// TIA Portal project "mixer" (V16)

(* hardware
DEVICE "S7300/ET200M station_1"  S7-300 station
   slot 0: "Rail_0"  Rail  6ES7 390-1***0-0AA0
   slot 2: "PLC_1"  CPU 312  6ES7 312-1AE13-0AB0  V2.6
      slot 0: "MPI interface_1"  X1
*)

// ===== PLC "PLC_1"  CPU 312 =====

VAR_GLOBAL   // PLC tag table "Default tag table"
   "C Start" AT %I0.0 : Bool;
   "C stop" AT %I0.1 : Bool;
   "C ON" AT %M0.0 : Bool;
   "Empty level switch I" AT %I0.4 : Bool;
   "In valve1" AT %Q0.0 : Bool;
   "Lvl of mat A" AT %I0.3 : Bool;
   "In valve2" AT %Q0.1 : Bool;
   "Lvl of mat B" AT %I0.2 : Bool;
   "Agitator-mix- moto" AT %Q0.2 : Bool;
   "Temp Sensor" AT %I0.5 : Bool;
   "Heater" AT %Q0.3 : Bool;
   "out valve" AT %Q0.4 : Bool;
END_VAR

ORGANIZATION_BLOCK "Main"   // OB1, LAD
TITLE = "Main Program Sweep (Cycle)"
{ S7_Optimized_Access := 'FALSE' }
VERSION : 0.1
   VAR_TEMP
      OB1_EV_CLASS : Byte;   // Bits 0-3 = 1 (Coming event), Bits 4-7 = 1 (Event class 1)
      OB1_SCAN_1 : Byte;   // 1 (Cold restart scan 1 of OB 1), 3 (Scan 2-n of OB 1)
      OB1_PRIORITY : Byte;   // Priority of OB Execution
      OB1_OB_NUMBR : Byte;   // 1 (Organization block 1, OB1)
      OB1_RESERVED_1 : Byte;   // Reserved for system
      OB1_RESERVED_2 : Byte;   // Reserved for system
      OB1_PREV_CYCLE : Int;   // Cycle time of previous OB1 scan (milliseconds)
      OB1_MIN_CYCLE : Int;   // Minimum cycle time of OB1 (milliseconds)
      OB1_MAX_CYCLE : Int;   // Maximum cycle time of OB1 (milliseconds)
      OB1_DATE_TIME : Date_And_Time;   // Date and time OB1 started
   END_VAR
BEGIN

REGION Network 1
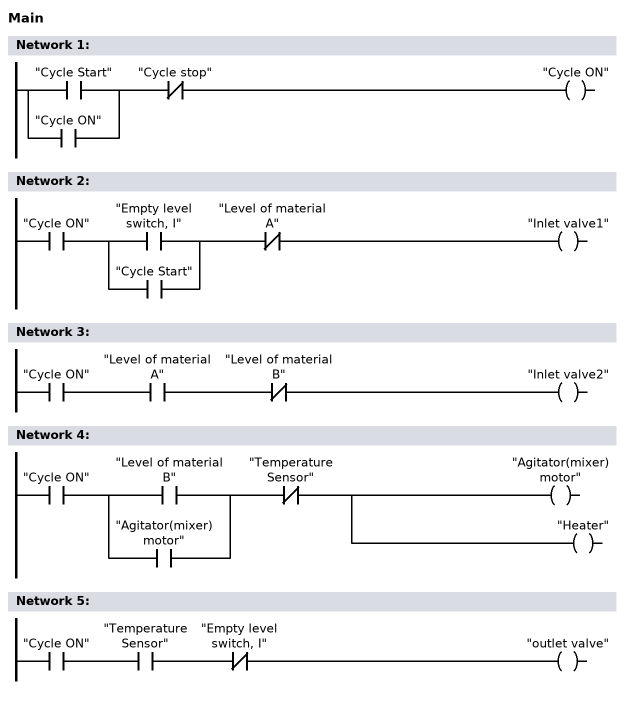
   RUNG wire#powerrail
      Contact( "Cycle Start" )
      wire#w1
      I_Contact( "Cycle stop" )
      Coil( "Cycle ON" )
   END_RUNG
   RUNG wire#powerrail
      Contact( "Cycle ON" )
   END_RUNG wire#w1
   // the same network as SCL:
   "Cycle ON" := ("Cycle Start" OR "Cycle ON") AND NOT "Cycle stop";
END_REGION

REGION Network 2
   RUNG wire#powerrail
      Contact( "Cycle ON" )
      wire#w1
      Contact( "Empty level switch, I" )
      wire#w2
      I_Contact( "Level of material A" )
      Coil( "Inlet valve1" )
   END_RUNG
   RUNG wire#w1
      Contact( "Cycle Start" )
   END_RUNG wire#w2
   // the same network as SCL:
   "Inlet valve1" := "Cycle ON" AND ("Empty level switch, I" OR "Cycle Start") AND NOT "Level of material A";
END_REGION

REGION Network 3
   RUNG wire#powerrail
      Contact( "Cycle ON" )
      Contact( "Level of material A" )
      I_Contact( "Level of material B" )
      Coil( "Inlet valve2" )
   END_RUNG
   // the same network as SCL:
   "Inlet valve2" := "Cycle ON" AND "Level of material A" AND NOT "Level of material B";
END_REGION

REGION Network 4
   RUNG wire#powerrail
      Contact( "Cycle ON" )
      wire#w1
      Contact( "Level of material B" )
      wire#w2
      I_Contact( "Temperature Sensor" )
      wire#w3
      Coil( "Agitator(mixer) motor" )
   END_RUNG
   RUNG wire#w1
      Contact( "Agitator(mixer) motor" )
   END_RUNG wire#w2
   RUNG wire#w3
      Coil( "Heater" )
   END_RUNG
   // the same network as SCL:
   "Agitator(mixer) motor" := "Cycle ON" AND ("Level of material B" OR "Agitator(mixer) motor") AND NOT "Temperature Sensor";
   "Heater" := "Agitator(mixer) motor";
END_REGION

REGION Network 5
   RUNG wire#powerrail
      Contact( "Cycle ON" )
      Contact( "Temperature Sensor" )
      I_Contact( "Empty level switch, I" )
      Coil( "outlet valve" )
   END_RUNG
   // the same network as SCL:
   "outlet valve" := "Cycle ON" AND "Temperature Sensor" AND NOT "Empty level switch, I";
END_REGION
END_ORGANIZATION_BLOCK